TYPE M1Tabs :
(
	OVERVIEW := 0,
    RADIAL := 1,
    AXIAL := 2,
    IO := 3,
    CONFIG := 4
);
END_TYPE

(* stored: Version 1.1.0.1, ProductVersion 3.1.4018.2
   DUT M1Tabs: Id {ce60cf3e-295d-46d3-a221-fcdee20d1614} *)
